// TIA Portal V18 export
FUNCTION_BLOCK "alm"   // FB4, LAD
{ S7_Optimized_Access := 'TRUE' }
VERSION : 0.1
// stored: AutoNumber true, IsIECCheckEnabled false, IsRetainMemResEnabled false, MemoryReserve 100, SetENOAutomatically false, UDAEnableTagReadback false
   VAR_INPUT
      alarm_input : Array[0..95] of Bool;
   END_VAR
   VAR_OUTPUT
      alarmreg_output : Array[0..95] of Bool;
   END_VAR
   VAR_IN_OUT
      alarm_ack : Array[0..95] of Bool;
      almreset_ons : Bool;
      fault_dipslay_reg : Int;
   END_VAR
   VAR
      i : Int;
      alarmregtemp : Array[0..95] of Bool;
      temp : Array[0..95] of Bool;
   END_VAR
   VAR_TEMP   // added for the SCL form of the ladder/FBD networks
      _w1 : Bool;
      _w2 : Bool;
      _w3 : Bool;
   END_VAR
BEGIN

REGION Network 1
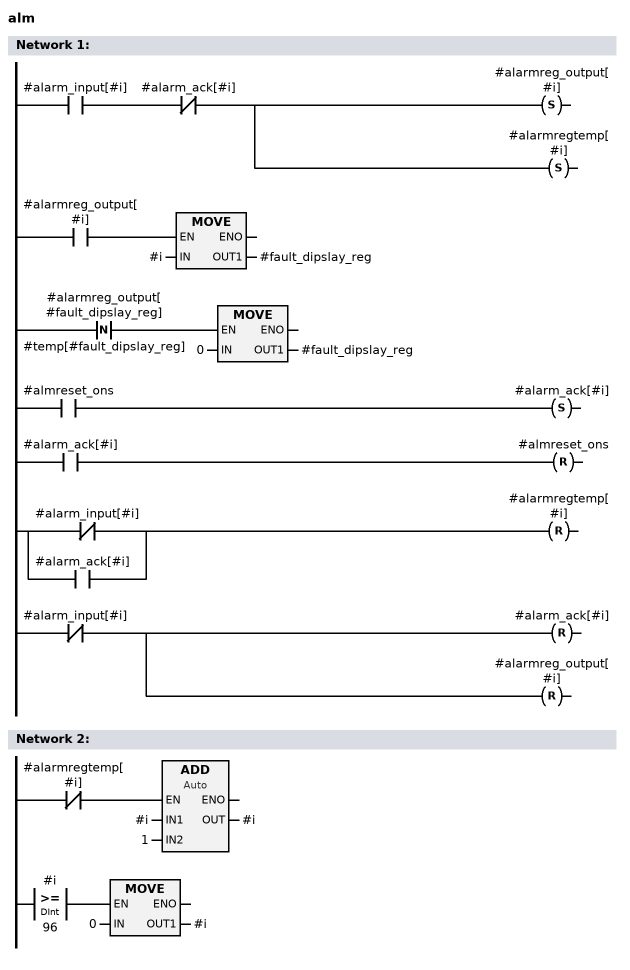
   RUNG wire#powerrail
      Contact( #alarm_input[#i] )
      I_Contact( #alarm_ack[#i] )
      wire#w1
      S_Coil( #alarmreg_output[#i] )
   END_RUNG
   RUNG wire#w1
      S_Coil( #alarmregtemp[#i] )
   END_RUNG
   RUNG wire#powerrail
      Contact( #alarmreg_output[#i] )
      Move(in := #i, out1 => #fault_dipslay_reg)
   END_RUNG
   RUNG wire#powerrail
      N_Contact(operand := #alarmreg_output[#fault_dipslay_reg], bit := #temp[#fault_dipslay_reg])
      Move(in := 0, out1 => #fault_dipslay_reg)
   END_RUNG
   RUNG wire#powerrail
      Contact( #almreset_ons )
      S_Coil( #alarm_ack[#i] )
   END_RUNG
   RUNG wire#powerrail
      Contact( #alarm_ack[#i] )
      R_Coil( #almreset_ons )
   END_RUNG
   RUNG wire#powerrail
      I_Contact( #alarm_input[#i] )
      wire#w2
      R_Coil( #alarmregtemp[#i] )
   END_RUNG
   RUNG wire#powerrail
      Contact( #alarm_ack[#i] )
   END_RUNG wire#w2
   RUNG wire#powerrail
      I_Contact( #alarm_input[#i] )
      wire#w3
      R_Coil( #alarm_ack[#i] )
   END_RUNG
   RUNG wire#w3
      R_Coil( #alarmreg_output[#i] )
   END_RUNG
   // the same network as SCL:
   #_w1 := #alarm_input[#i] AND NOT #alarm_ack[#i];
   IF #_w1 THEN
       #alarmreg_output[#i] := TRUE;
       #alarmregtemp[#i] := TRUE;
   END_IF;
   IF #alarmreg_output[#i] THEN #fault_dipslay_reg := #i; END_IF;
   #_w2 := NOT #alarmreg_output[#fault_dipslay_reg] AND #temp[#fault_dipslay_reg];   // falling edge of #alarmreg_output[#fault_dipslay_reg]
   #temp[#fault_dipslay_reg] := #alarmreg_output[#fault_dipslay_reg];
   IF #_w2 THEN #fault_dipslay_reg := 0; END_IF;
   IF #almreset_ons THEN #alarm_ack[#i] := TRUE; END_IF;
   IF #alarm_ack[#i] THEN #almreset_ons := FALSE; END_IF;
   IF NOT #alarm_input[#i] OR #alarm_ack[#i] THEN #alarmregtemp[#i] := FALSE; END_IF;
   #_w3 := NOT #alarm_input[#i];
   IF #_w3 THEN
       #alarm_ack[#i] := FALSE;
       #alarmreg_output[#i] := FALSE;
   END_IF;
END_REGION

REGION Network 2
   RUNG wire#powerrail
      I_Contact( #alarmregtemp[#i] )
      Add(in1 := #i, in2 := 1, out => #i)
   END_RUNG
   RUNG wire#powerrail
      { S7_Templates := "SrcType := DInt" } GE_Contact(in1 := #i, in2 := 96)
      Move(in := 0, out1 => #i)
   END_RUNG
   // the same network as SCL:
   IF NOT #alarmregtemp[#i] THEN #i := #i + 1; END_IF;
   IF #i >= 96 THEN #i := 0; END_IF;
END_REGION
END_FUNCTION_BLOCK
